Staubli VAL3: example.pgx

program example()
  local num l_nLanguage
begin
  //-----------------------------------------------------------------------
  //Header begin
  //Description of program
  //  This is an example for use this library.
  //  This program run differents sub-programs :
  //  - language() for choose the language : "English or "Deutsch"
  //  - aMainTcp() for calculates the tool transformation : a wizard will
  //  guide you thtough the steps.
  //
  //Traceability
  //  Creation : 08-04-08 - f.Rob
  //Header end
  //-----------------------------------------------------------------------

  call language()
  call aMainTcp(nLangSet)
end
